{attribute addProperty BoxType "ELX3204-0000-0016"}
{attribute addProperty Id "RTD_Inputs_ChannelAT %I*ARRAY[0..6] OF RTD_Inputs_Channel_F16A160D128160WcStateAT %I*WcState_98A4DF7520.250InfoDataAT %I*InfoData_BC63D37F80100"}
{attribute addProperty CRC "647171617"}
{attribute addProperty SizeInBites "210"}
{attribute addProperty SizeInBytes "26.25"}
TYPE ELX3204_B9E43530 :
STRUCT
	{attribute addProperty Name "RTD_Inputs_Channel"}
	RTD_Inputs_Channel : ARRAY[0..6] OF RTD_Inputs_Channel_F16A160D;
	{attribute addProperty Name "WcState"}
	WcState : WcState_98A4DF75;
	{attribute addProperty Name "InfoData"}
	InfoData : InfoData_BC63D37F;
END_STRUCT
END_TYPE

(* stored: Version 1.2.0.0, ProductVersion 3.1.4024.9
   DUT ELX3204_B9E43530: Id {dea95d06-c733-4274-8422-90c38b86f71b} *)
